
DATA_BLOCK DB303
    STRUCT
        LEITURA: ARRAY[0 .. 102] OF WORD;
    END_STRUCT
BEGIN
END_DATA_BLOCK
